FUNCTION_BLOCK HydroGenerateSessionKeyServer (* Service Interface Function Block Type *)
  (* Standard: 61499-2 *)
  (* Version 1.0, 2019-11-18, Awais *)
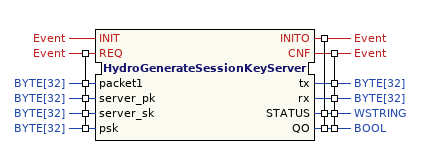
  EVENT_INPUT
    INIT; (* Service Initialization *)
    REQ WITH server_sk, server_pk, packet1, psk; (* Service Request *)
  END_EVENT
  EVENT_OUTPUT
    INITO WITH QO, STATUS; (* Initialization Confirm *)
    CNF WITH QO, STATUS, tx, rx; (* Confirmation of Requested Service *)
  END_EVENT
  VAR_INPUT
    packet1 : ARRAY [0..31] OF BYTE := 0; (* packet recieved from the client. *)
    server_pk : ARRAY [0..31] OF BYTE := 0; (* Server public key *)
    server_sk : ARRAY [0..31] OF BYTE := 0; (* Server secret key (must not be communicated) *)
    psk : ARRAY [0..31] OF BYTE := 0; (* pre-shared secret *)
  END_VAR
  VAR_OUTPUT
    tx : ARRAY [0..31] OF BYTE := 0; (* Key for sending data to the client, *)
    rx : ARRAY [0..31] OF BYTE := 0; (* Key for receiving data from the client *)
    STATUS : WSTRING; (* Service Status *)
    QO : BOOL; (* Event Output Qualifier *)
  END_VAR
  SERVICE APPLICATION/RESOURCE (* Service Interface Function Block Type *)
    SEQUENCE normal_establishment
      APPLICATION.INIT+(PARAMS) -> RESOURCE.initialize(PARAMS) -> APPLICATION.INITO+();
    END_SEQUENCE
    SEQUENCE unsuccessful_establishment
      APPLICATION.INIT+(PARAMS) -> RESOURCE.initialize(PARAMS) -> APPLICATION.INITO-(STATUS);
    END_SEQUENCE
    SEQUENCE request_confirm
      APPLICATION.REQ+(SD) -> RESOURCE.request(SD) -> APPLICATION.CNF+(RD);
    END_SEQUENCE
    SEQUENCE request_inhibited
      APPLICATION.REQ-(SD) -> APPLICATION.CNF-(STATUS);
    END_SEQUENCE
    SEQUENCE request_error
      APPLICATION.REQ+(SD) -> RESOURCE.request(SD) -> APPLICATION.CNF-(STATUS);
    END_SEQUENCE
    SEQUENCE indication_response
      RESOURCE.indicate(RD) -> APPLICATION.IND+(RD);
      APPLICATION.RSP(QI,SD) -> RESOURCE.response(QI,SD);
    END_SEQUENCE
    SEQUENCE indication_inhibited
      RESOURCE.indicate(RD,QI=FALSE) -> RESOURCE.inhibited();
    END_SEQUENCE
    SEQUENCE error_indication
      RESOURCE.error(STATUS) -> APPLICATION.IND-(STATUS);
    END_SEQUENCE
    SEQUENCE application_initiated_termination
      APPLICATION.INIT-() -> RESOURCE.terminate() -> APPLICATION.INITO-(STATUS);
    END_SEQUENCE
    SEQUENCE resource_initiated_termination
      -> APPLICATION.INITO-(STATUS);
    END_SEQUENCE
  END_SERVICE
END_FUNCTION_BLOCK
